{attribute 'qualified_only'}
{attribute 'strict'}
TYPE E_OpMode :
(
	Stop,
	Manual, 
	Jog,
	Automatic,
	AutomaticRunning
);
END_TYPE

(* stored: Version 1.1.0.1, ProductVersion 3.1.4024.11
   DUT E_OpMode: Id {5701ba74-657b-4cae-b91f-d981ee74d4ad} *)
